Fanuc KAREL source: wmotype.kl

PROGRAM wmotype
%NOLOCKGROUP
VAR
  p : POSITION
  q : POSITION
  i : INTEGER
  r : REAL
BEGIN
  WITH $MOTYPE = LINEAR MOVE TO p
END wmotype
